Universal Robots PolyScope program: Pallet2.urp

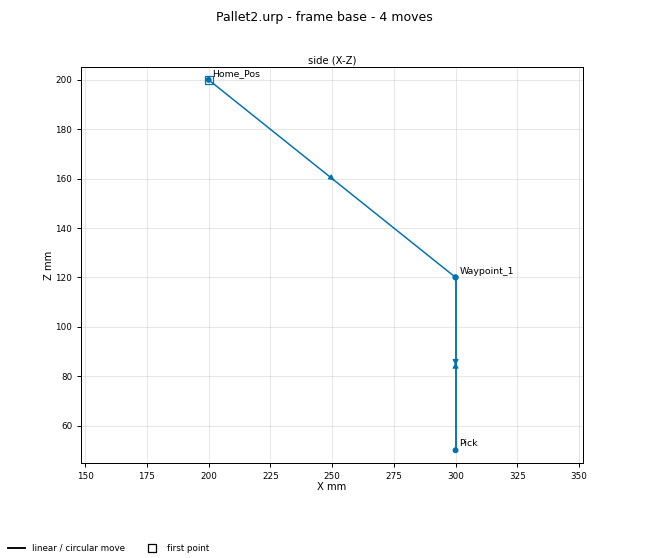
[picture p0: tool path of Pallet2.urp in frame base, 4 of 4 moves have a stored position in this frame; points joined in program order, loops and branches not executed]
Program Pallet2 (installation=default directory=/home/ur/ursim-current/programs createdIn=3.15.6.106324 lastSavedIn=3.15.6.106324 robotSerialNumber=2018339999)
Calibrated DH parameters: a=[0, -0.24365, -0.21325, 0, 0, 0]; d=[0.1519, 0, 0, 0.11235, 0.08535, 0.0819]; alpha=[1.570796, 0, 0, 1.570796, -1.570796, 0]; deltaTheta=[0, 0, 0, 0, 0, 0]
Robot Program (runOnlyOnce=true)
  MoveJ speed 60 deg/s, acceleration 80 deg/s^2 (useActiveTCP=true)
    Waypoint Home_Pos: TCP in base x=200 y=200 z=200 mm, rx=3.14 ry=0 rz=0 rad; joints [68.428, -80.897, -101.913, -87.275, 89.966, -21.572] deg; flange x=200 y=200.159 z=300 mm, rx=3.14 ry=0 rz=0 rad
  Set DigitalOutput pin=digital_out[2]; digitalValue=0
  Wait DigitalInput pin=Sensor; digitalValue=1
  Loop Counting (count=27) loopVariable(name=Loop_2)
    MoveL speed 250 mm/s, acceleration 500 mm/s^2 (useActiveTCP=true) feature=Base
      Waypoint Waypoint_1: TCP in base x=300 y=200 z=120 mm, rx=3.14 ry=0 rz=0 rad; joints [51.876, -104.758, -98.881, -66.433, 89.944, -38.124] deg; flange x=300 y=200.159 z=220 mm, rx=3.14 ry=0 rz=0 rad
      Waypoint Pick: TCP in base x=300 y=200 z=50 mm, rx=3.14 ry=0 rz=0 rad; joints [51.876, -113.936, -108.026, -48.109, 89.944, -38.124] deg; flange x=300 y=200.159 z=150 mm, rx=3.14 ry=0 rz=0 rad
      Set DigitalOutput pin=digital_out[0]; digitalValue=1
      Wait Sleep waitTime=0.3
      Waypoint Waypoint_1: TCP in base x=300 y=200 z=120 mm, rx=3.14 ry=0 rz=0 rad; joints [51.876, -104.758, -98.881, -66.433, 89.944, -38.124] deg; flange x=300 y=200.159 z=220 mm, rx=3.14 ry=0 rz=0 rad
      Pallet pattern(dimensionality=Box firstAxisCount=3 secondAxisCount=3 thirdAxisCount=3 motionType=MoveL speed=0.25 acceleration=1.2 useActiveTCP=true, counterVariable(name=cnt_3, initializeExpression=0), patternPoseVariable(name=pose_3), feature=Base, children(Waypoint(type=Fixed name=Corner1_3, position(joints=-0.14375859895815069, -1.7459991613971155, -2.243671719227926, -0.7224891821490687, 1.569219946861267, -1.7145550886737269 pose=0.25000005555105786, -0.15000006073029226, 0.05000000291213959, 3.1399997393831147, -2.7168847606307495E-8, 1.126408290855774E-6), poseInFeatureCoordinates=[0.25, -0.15, 0.05, 3.14, 0, 0.000001], outputFlangePose=[0.25, -0.149841, 0.15, 3.14, 0, 0.000001]), Waypoint(type=Fixed name=Corner2_3, position(joints=-0.10459643999208623, -2.0563228766070765, -1.773836914693014, -0.8820622603045862, 1.5692121982574463, -1.6753929297076624 pose=0.3500000122261205, -0.14999997530905035, 0.04999993337458872, 3.1399997545626834, 4.852446761243972E-8, 9.795029553284414E-7), poseInFeatureCoordinates=[0.35, -0.15, 0.05, 3.14, 0, 0.000001], outputFlangePose=[0.35, -0.149841, 0.15, 3.14, 0, 0.000001]), Waypoint(type=Fixed name=Corner3_3, position(joints=-0.355321232472555, -2.2277515570269983, -1.472224537526266, -1.0118582884417933, 1.5693031549453735, -1.9261181990252894 pose=0.3500000218679246, -0.24999995954696896, 0.04999989209936778, 3.139999813633263, 3.5467553023354856E-7, 7.720648011757946E-7), poseInFeatureCoordinates=[0.35, -0.25, 0.05, 3.14, 0, 0.000001], outputFlangePose=[0.35, -0.249841, 0.15, 3.14, 0, 0.000001]), Waypoint(type=Fixed name=Corner4_3, position(joints=-0.46124345461000615, -1.964156452809469, -1.9257891813861292, -0.8217342535602015, 1.569370150566101, -2.0320408979998987 pose=0.24999999428034708, -0.2499999619187932, 0.05000003462183589, 3.1399999233202416, 9.595120886328885E-7, 3.9946142311507015E-7), poseInFeatureCoordinates=[0.25, -0.25, 0.05, 3.14, 0.000001, 0], outputFlangePose=[0.25, -0.249841, 0.15, 3.14, 0.000001, 0]), Waypoint(type=Fixed name=Corner5_3, position(joints=-0.14375859895815069, -1.4585326353656214, -1.834332291279928, -1.419295612965719, 1.5692200660705566, -1.7145550886737269 pose=0.2499999150938191, -0.1500000185148824, 0.18000004132238367, 3.13999992567651, -2.6557426762175424E-8, 4.1230966185074084E-7), poseInFeatureCoordinates=[0.25, -0.15, 0.18, 3.14, 0, 0], outputFlangePose=[0.25, -0.149841, 0.28, 3.14, 0, 0]), Waypoint(type=Fixed name=Corner6_3, position(joints=-0.10459643999208623, -1.847318474446432, -1.4089844862567347, -1.4559195677386683, 1.5692123174667358, -1.6753929297076624 pose=0.3500000234020807, -0.14999995470580527, 0.17999999488259819, 3.1399999229052358, 4.91329434437926E-8, 2.545005611053244E-7), poseInFeatureCoordinates=[0.35, -0.15, 0.18, 3.14, 0, 0], outputFlangePose=[0.35, -0.149841, 0.28, 3.14, 0, 0]), Waypoint(type=Fixed name=Corner7_3, position(joints=-0.355321232472555, -2.069094959889547, -1.0915792624102991, -1.5511601606952112, 1.5693031549453735, -1.9261181990252894 pose=0.3500000692875774, -0.24999997717144573, 0.18000008977980203, 3.1399998136333327, 3.5467557020129767E-7, 7.720648558910128E-7), poseInFeatureCoordinates=[0.35, -0.25, 0.18, 3.14, 0, 0.000001], outputFlangePose=[0.35, -0.249841, 0.28, 3.14, 0, 0.000001]), Waypoint(type=Fixed name=Corner8_3, position(joints=-0.46124345461000615, -1.7299845854388636, -1.5557406584369105, -1.4259541670428675, 1.569370150566101, -2.0320404211627405 pose=0.25000002328574644, -0.2499999763642055, 0.18000018583891197, 3.139999711098197, 2.1034396716191406E-7, 1.0704594441409317E-6), poseInFeatureCoordinates=[0.25, -0.25, 0.18, 3.14, 0, 0.000001], outputFlangePose=[0.25, -0.249841, 0.28, 3.14, 0, 0.000001]))); actionSequence(name=PalletSequence motionType=MoveL speed=0.25 acceleration=1.2 useActiveTCP=true, anchorWaypoint(type=Fixed name=PatternPlace, position(joints=-0.27030831972231084, -1.7601545492755335, -1.5194199720965784, -1.4323895613299769, 1.5692615509033203, -1.8411052862750452 pose=0.3000000643323511, -0.20000004406723254, 0.1799999570512242, 3.1400001480158486, 4.928250918857606E-7, -5.662763665721766E-7), poseInFeatureCoordinates=[0.3, -0.2, 0.18, 3.14, 0, -0.000001], outputFlangePose=[0.3, -0.199841, 0.28, 3.14, 0, -0.000001]), feature=Base, children(Waypoint(type=Fixed name=Approach, position(joints=-0.27030831972231084, -1.768360439931051, -1.1795113722430628, -1.764092270527975, 1.5692615509033203, -1.8411052862750452 pose=0.300000040449905, -0.20000003746454137, 0.24999998889583266, 3.140000148015988, 4.928250655378751E-7, -5.662762571188324E-7), poseInFeatureCoordinates=[0.3, -0.2, 0.25, 3.14, 0, -0.000001], outputFlangePose=[0.3, -0.199841, 0.35, 3.14, 0, -0.000001]), Waypoint=PatternPlace, Set(type=DigitalOutput, pin=digital_out[0], digitalValue=0), Wait(type=Sleep, waitTime=0.3), Waypoint(type=Fixed name=Exit_, position(joints=-0.27030831972231084, -1.768360439931051, -1.1795113722430628, -1.764092270527975, 1.5692615509033203, -1.8411052862750452 pose=0.300000040449905, -0.20000003746454137, 0.24999998889583266, 3.140000148015988, 4.928250655378751E-7, -5.662762571188324E-7), poseInFeatureCoordinates=[0.3, -0.2, 0.25, 3.14, 0, -0.000001], outputFlangePose=[0.3, -0.199841, 0.35, 3.14, 0, -0.000001])))
        Pattern -> pattern
        AnchoredSequence -> PalletSequence
  Set DigitalOutput pin=digital_out[2]; digitalValue=1
